PROGRAM MAIN
VAR
	fbPower: FB_PowerChannel;
	runGCode: ItpEnableDefaultGCode;
	fbBuildGroup: CfgBuildExt3DGroup;
	fbLoadGCode: ItpLoadProgEx;
	fbStartGCode: ItpStartStopEx;
	fbConfirmHsk: ItpConfirmHsk;
	getSParam :ItpGetSParam;
	
	Xaxis: AXIS_REF;
	Yaxis: AXIS_REF;
	Zaxis: AXIS_REF;
	Extruder: AXIS_REF;

	Xhome: MC_Home;
	Yhome: MC_Home;
	Zhome: MC_Home;
	
	HomingSensorX: BOOL;
	HomingSensorY: BOOL;
	HomingSensorZ: BOOL;
	
	
	in_stNciToPlc AT %I*: NCTOPLC_NCICHANNEL_REF;
	out_stPlcToNci AT %Q*: PLCTONC_NCICHANNEL_REF;
	
	
	State: INT;
	bConfirmHsk: BOOL := FALSE;
	sPrgName: STRING(255) := 'test.txt';
	nInterpreterState: UDINT;
	
END_VAR


fbPower(
	bEnable:=TRUE, 
	fOvr:= 100.0, 
	stX:=Xaxis, 
	stY:=Yaxis, 
	stZ:=Zaxis, 
	stPlcToNci:=out_stPlcToNci , 
	bAllAxesReady=> );
	

	
CASE State OF
	0: // init
	
	IF fbPower.bAllAxesReady THEN
		State := 20; 
	END_IF
	
	10:
	
	Xhome(axis := Xaxis,execute := TRUE,BCalibrationCam := HomingSensorX);
	IF Xhome.Done THEN
		State:=11;
	END_IF
	
	11:
	
	Yhome(axis := Yaxis,execute := TRUE,BCalibrationCam := HomingSensorY);
	IF Xhome.Done THEN
		State:=12;
	END_IF
	
	12:
	
	Zhome(axis := Zaxis,execute := TRUE,BCalibrationCam := HomingSensorZ);
	IF Zhome.Done THEN
		State:=12;
	END_IF
	
	20:
	
	fbBuildGroup(
		bExecute:=TRUE,
		nGroupId:=ItpGetGroupId(sNciToPlc:=in_stNciToPlc),
		nXAxisId:=XAxis.NcToPlc.AxisId,
		nYAxisId:=YAxis.NcToPlc.AxisId,
		nZAxisId:=ZAxis.NcToPlc.AxisId,
		tTimeOut:=t#2s );
	IF NOT fbBuildGroup.bBusy THEN
		fbBuildGroup( bExecute:=FALSE );
		(* error handling missing *)
		State	:= 30;
	END_IF
	
	30:
	
	fbLoadGCode(
		sNciToPlc:=in_stNciToPlc, 
		bExecute:=TRUE, 
		sPrg:= sPrgName, 
		nLength:= INT_TO_UDINT(LEN(sPrgName)), 
		tTimeOut:= , 
		bBusy=> , 
		bErr=> , 
		nErrId=> );
	IF NOT fbLoadGCode.bBusy THEN
		IF NOT fbLoadGCode.bErr THEN
			State	:= 40;				
		END_IF
		fbLoadGCode(sNciToPlc:=in_stNciToPlc, bExecute:=FALSE); 
	END_IF
	40:
	
	nInterpreterState	:= ItpGetStateInterpreter(sNciToPlc:=in_stNciToPlc);
	IF nInterpreterState = Tc2_NCI.NCI_INTERPRETER_READY THEN
		State	:= 50;		
	END_IF
	50:
	
	// start g-code file
	fbStartGCode(
		bStart:=TRUE, 
		bStop:=FALSE, 
		tTimeOut:= , 
		sNciToPlc:= in_stNciToPlc, 
		bBusy=> , 
		bErr=> , 
		nErrId=> );
	IF NOT fbStartGCode.bBusy THEN
		IF NOT fbStartGCode.bErr THEN
			State	:= 60;			
		END_IF
		fbStartGCode( bStart:=FALSE, sNciToPlc:= in_stNciToPlc ); 
	END_IF
	60: 
	
	
END_CASE


IF ItpIsHskMFunc(in_stNciToPlc) AND NOT fbConfirmHsk.bBusy THEN
	bConfirmHsk	:= TRUE;
ELSE	
	bConfirmHsk	:= FALSE;
END_IF	

fbConfirmHsk(
	bExecute:=bConfirmHsk , 
	sNciToPlc:=in_stNciToPlc , 
	sPlcToNci:=out_stPlcToNci , 
	bBusy=> , 
	bErr=> , 
	nErrId=> );

END_PROGRAM

(* stored: Version 1.1.0.1, ProductVersion 3.1.4024.9
   POU MAIN: Id {7d554d0f-1162-429d-8d78-ee6190d9367c}, SpecialFunc None *)
